FUNCTION RAD_TO_DEG : LREAL
VAR_INPUT
    rad : LREAL;
END_VAR
VAR
END_VAR

RAD_TO_DEG := rad * 180.0 / PI;

END_FUNCTION

(* stored: Version 1.1.0.1, ProductVersion 3.1.4018.5
   POU RAD_TO_DEG: Id {ece4e8f5-8083-47bd-b4d1-3b5cc440820e}, SpecialFunc None *)
